FUNCTION_BLOCK "LGF_TimerSwitch"
{ S7_Optimized_Access := 'TRUE' }
VERSION : 0.1
   VAR_INPUT
      onMonth : USInt;   // Monat, in der der Ausgang gesetzt wird
      onDay : USInt;   // Tag, an dem der Ausgang gesetzt wird
      onWeekday : USInt;   // Wochentag, an dem der Ausgang gesetzt wird;  Sonntag: 1, Montag: 2, Dienstag: 3, ...
      onHour : USInt;   // Stunde, in der der Ausgang gesetzt wird
      onMinute : USInt;   // Minute, in der der Ausgang gesetzt wird
      offMonth : USInt;   // Monat, in der der Ausgang zurückgesetzt wird
      offDay : USInt;   // Tag, an dem der Ausgang zurückgesetzt wird
      offWeekday : USInt;   // Wochentag, an dem der Ausgang zurückgesetzt wird;  Sonntag: 1, Montag: 2, Dienstag: 3, ...
      offHour : USInt;   // Stunde, in der der Ausgang zurückgesetzt wird
      offMinute : USInt;   // Minute, in der der Ausgang zurückgesetzt wird
      mode : USInt;   // Angabe des Modus (siehe Funktionsweise);  Täglich: 1, Wöchentlich: 2, Monatlich: 3, Jährlich: 4, Arbeitstage: 5, Wochenende: 6
   END_VAR

   VAR_OUTPUT
      signal { ExternalWritable := 'False'} : Bool;   // Ausagngssignal
      actLocalTime {InstructionName := 'DTL'; LibVersion := '1.0'; ExternalWritable := 'False'} : DTL;   // Aktuelle Lokalzeit
      error { ExternalWritable := 'False'} : Bool;   // FALSE: Kein Fehler / TRUE: Während der Ausführung des FB ist ein Fehler aufgetreten
      status { ExternalWritable := 'False'} : Word;   // 16#0000-16#7FFF: Status des FB / 16#8000-16#FFFF: Fehleridentifikation (siehe folgende Tabelle)
      subFunctionStatus { ExternalWritable := 'False'} : Word;   // Status Word einer aufgerufenen Unterfunktion
   END_VAR

   VAR_TEMP
      tempTime {InstructionName := 'DTL'; LibVersion := '1.0'} : DTL;   // Temp Variable für die aktuelle Zeit und das aktuelle Datum von RD_LOC_T
      tempReadTimeStatus : Word;   // Status Wort der Systemfunktion RD_LOC_T
      tempOnTimeDtl {InstructionName := 'DTL'; LibVersion := '1.0'} : DTL;   // Temp Variable für Einschaltzeitpunkt (Zeit und Datum) DTL
      tempOnTimeTod : Time_Of_Day;   // Temp Variable für Einschaltzeitpunkt (Zeit) TOD
      tempOffTimeDtl {InstructionName := 'DTL'; LibVersion := '1.0'} : DTL;   // Temp Variable für Ausschaltzeitpunkt (Zeit und Datum) DTL
      tempOffTimeTod : Time_Of_Day;   // Temp Variable für Ausschaltzeitpunkt (Zeit) TOD
      tempActTimeDtl {InstructionName := 'DTL'; LibVersion := '1.0'} : DTL;   // Temp Variable für aktuelles Datum und aktuelle Zeit DTL
      tempActTimeTod : Time_Of_Day;   // Temp Variable für aktuelles Datum und aktuelle Zeit von RD_LOC_T / TOD
   END_VAR

   VAR CONSTANT
      ZERO : USInt := 0;   // Null Konstante zur Initialisierung
      CLEAR_DTL {InstructionName := 'DTL'; LibVersion := '1.0'} : DTL;   // Lösche Datum und Zeit mit leerer Varibale
      STATUS_NO_ERROR : Word := 16#0000;   // Status: kein Fehler aufgetreten
      ERR_NO_MODE_SELECTED : Word := 16#8200;   // Error: Kein vorhandener Mode ausgewählt, bitte Eingang `mode` prüfen
      ERR_RD_LOC_T : Word := 16#8600;   // Error in Funktion RD_LOC_T - weitere infos in `subFunctionStatus`
      MODE_DAILY : UInt := 1;   // Mode: Täglich
      MODE_WEEKLY : UInt := 2;   // Mode: Wöchentlich
      MODE_MONTHLY : UInt := 3;   // Mode: Monatlich
      MODE_YEARLY : UInt := 4;   // Mode: Jährlich
      MODE_WEEK_DAYS : UInt := 5;   // Mode: Wochentage
      MODE_WEEKEND_DAYS : UInt := 6;   // Mode: Wochenend Tage
      MONTH_JANUARY : USInt := 1;   // Monat Januar
      MONTH_DECEMBER : USInt := 12;   // Monat Dezember
      DAY_MONDAY : USInt := 2;   // Wochentag Montag
      DAY_FRIDAY : USInt := 6;   // Wochentag Freitag
      DAY_SATURDAY : USInt := 7;   // Wochentag Samstag
      DAY_SUNDAY : USInt := 1;   // Wochentag Sonntag
      DAY_NEXT_SUNDAY : USInt := 8;   // Wochentag - mächster Sonntag
      DAY_NEXT_MONDAY : USInt := 9;   // Wochentag - nächster Montag
      DATE_INCREMENT : USInt := 1;   // Inkremntierung für Datum (Monat oder Jahr)
      DAY_INCREMENT : Time := T#1d;   // Inkrementiere einen Tag
      WEEK_INCREMENT : Time := T#7d;   // Inkremntiere 7 Tage = 1 Woche
      DAYS_PER_WEEK : USInt := 7;   // Eine Woche = 7 Tage
      DEFAULT_YEAR : UInt := 2015;   // Default Jahr um im DTL Datentyp den Wochentag und das Datum zu synchronisieren
      DEFAULT_MONTH : USInt := 2;   // Default Monat um im DTL Datentyp den Wochentag und das Datum zu synchronisieren
   END_VAR


BEGIN
	REGION BLOCK INFO HEADER
	    //===============================================================================
	    // SIEMENS AG / (c)Copyright 2017
	    //-------------------------------------------------------------------------------
	    // Title:            LGF_TimerSwitch
	    // Comment/Function: Timer Switch (daily, weekly, monthly, working days, ...)
	    //                   Mode: Daily: 1, weekly: 2, monthly: 3, yearly: 4, workday: 5, weekend: 6
	    // Library/Family:   LGF(Library General Functions)
	    // Author:           Siemens Digital Industry Support
	    // Tested with:      CPU1212C DC/DC/DC FW:V4.2
	    // Engineering:      TIA Portal V14 Update 1
	    // Restrictions:     ENO disabled - error handling done with error and status
	    // Requirements:     PLC (S7-1200 / S7-1500)
	    //-------------------------------------------------------------------------------
	    // Change log table:
	    // Version  | Date       | Expert in charge       | Changes applied
	    //----------|------------|------------------------|------------------------------
	    // 01.00.00 19.08.2015  Siemens Industry Online Support
	    //                      First released version
	    // 01.00.01 16.11.2015  Siemens Industry Online Support
	    //                      Fix in mode 2
	    // 01.01.00 23.05.2016  Siemens Industry Online Support
	    //                      New mode 5 + 6
	    //                      New output: actLocalTime
	    // 01.01.01 02.01.2017  Siemens Industry Online Support
	    //                      Upgrade: TIA V14 Update 1
	    // 01.01.02 14.09.2018  Siemens Industry Online Support
	    //                      Fix in modes 1, 3, 5, 6
	    // 01.01.03 17.09.2018  Siemens Industry Online Support
	    //                      Upgrade: TIA V15 Update 2
	    // 01.01.04 10.10.2018  Siemens Industry Online Support
	    //                      Connection to type restored
	    // 01.01.05 23.11.2018  Siemens Industry Online Support
	    //                      Upgrade: TIA V15.1
	    // 01.01.10 13.11.2019  Simatic Systems Support
	    //                      Magic numbers removed, tag naming added, code reworked
	    // 03.00.00 23.04.2020  Simatic Systems Support
	    //                      Set version to V3.0.0, harmonize the version of the whole library
	    // 03.00.01 19.01.2020  Simatic Systems Support
	    //                      Insert documentation
	    //=============================================================================
	END_REGION BLOCK INFO HEADER

	REGION DESCRIPTION
	    (/*
	Hinweis
	:    In `subFunctionStatus` wird der Status von aufgerufenen Anweisungen ausge-geben. Der Ausgangswert in `status` gibt in diesem Fall an, welche Anweisung den Fehler verursacht hat. Holen Sie sich in diesem Fall die Informationen aus der TIA Portal Online Hilfe zu den jeweiligen Anweisungen.

	---

	Der Baustein bietet verschiedene Arten einer Zeitschaltuhr, die im Parameter `mode` bestimmt werden

	* Tägliche Zeitschaltuhr (mode = 1)
	* Wöchentliche Zeitschaltuhr (mode = 2)
	* Monatliche Zeitschaltuhr (mode = 3)
	* Jährliche Zeitschaltuhr (mode = 4)
	* Werktags, Montag bis Freitag (mode = 5)
	* Wochenende, Samstag und Sonntag (mode = 6)

	Der Zeitwert wird immer mit der Lokalzeit der SPS verglichen, daher muss der Zeitwert, der bei den On- und Off-Parametern angegeben wird, als lokale Zeit angegeben werden.

	Abhängig vom Modus müssen folgende Formalparameter beschaltet werden:

	+------+---------------------------------------+-----------------------------------------+
	| Mode | Mode                                  | Required formal parameters              |
	+======+=======================================+=========================================+
	| 1 .  | Tägliche Zeitschaltuhr                | * onHour / offHour                      |
	|      |                                       | * onMinute / offMinute                  |
	+------+---------------------------------------+-----------------------------------------+
	| 2 .  | Wöchentlich Zeitschaltuhr             | * onWeekday / offWeekday                |
	|      |                                       | * onHour / offHour                      |
	|      |                                       | * onMinute / offMinute                  |
	+------+---------------------------------------+-----------------------------------------+
	| 3 .  | Monatliche Zeitschaltuhr              | * onDay / offDay                        |
	|      |                                       | * onHour / offHour                      |
	|      |                                       | * onMinute / offMinute                  |
	+------+---------------------------------------+-----------------------------------------+
	| 4 .  | Jährliche Zeitschaltuhr               | * onMonth / offMonth                    |
	|      |                                       | * onDay / offDay                        |
	|      |                                       | * onHour / offHour                      |
	|      |                                       | * onMinute / offMinute                  |
	+------+---------------------------------------+-----------------------------------------+
	| 5 .  | Werktags                              | * onHour / offHour                      |
	|      |                                       | * onMinute / offMinute                  |
	+------+---------------------------------------+-----------------------------------------+
	| 6 .  | Wochenende                            | * onHour / offHour                      |
	|      |                                       | * onMinute / offMinute                  |
	+------+---------------------------------------+-----------------------------------------+

	Entspricht die eingestellte Startzeit der aktuellen Lokalzeit der Steuerung, wird der Ausgang `signal` auf `TRUE` gesetzt. Entspricht die eingestellte Abschaltzeit der aktuellen Lokalzeit der Steuerung, wird der Ausgang `signal` wieder zurückgesetzt.

	Hinweis
	:    Beachten Sie, dass der Baustein in den Modi „Monatliche Zeitschaltuhr“ (mode = 3) oder „Jährliche Zeitschaltuhr“ (mode = 4) nur dann schaltet, wenn die Tage, die Sie an den Eingangsparametern „onDay“ und „offDay“ angeben, tatsächlich in diesem Monat vorkommen.
	*/)
	END_REGION DESCRIPTION

	REGION INITIALISATION
	    // Time ON init
	    #tempOnTimeDtl.HOUR := #onHour;
	    #tempOnTimeDtl.MINUTE := #onMinute;
	    #tempOnTimeDtl.SECOND := #ZERO;
	    #tempOnTimeDtl.NANOSECOND := #ZERO;
	    // Time OFF init
	    #tempOffTimeDtl.HOUR := #offHour;
	    #tempOffTimeDtl.MINUTE := #offMinute;
	    #tempOffTimeDtl.SECOND := #ZERO;
	    #tempOffTimeDtl.NANOSECOND := #ZERO;
	END_REGION

	REGION READ LOCAL TIME
	    #tempReadTimeStatus := INT_TO_WORD(RD_LOC_T(#tempTime));

	    // check result for error --> 16#8000 / MSB .X15
	    IF #tempReadTimeStatus.%X15 THEN
	        #error := TRUE;
	        #status := #ERR_RD_LOC_T;
	        #subFunctionStatus := #tempReadTimeStatus;
	        #actLocalTime := #CLEAR_DTL;
	        #signal := FALSE;
	        RETURN;
	    END_IF;

	    // Store time of the current day
	    #tempActTimeDtl := #tempTime;
	    #tempActTimeTod := DTL_TO_TOD(#tempTime);
	END_REGION

	REGION TIMER SWITCH LOGIC
	    CASE #mode OF
	        #MODE_DAILY:
	            REGION DAILY MODE
	                #tempOnTimeDtl.YEAR := #tempActTimeDtl.YEAR;
	                #tempOnTimeDtl.MONTH := #tempActTimeDtl.MONTH;
	                #tempOnTimeDtl.WEEKDAY := #tempActTimeDtl.WEEKDAY;
	                #tempOnTimeDtl.DAY := #tempActTimeDtl.DAY;
	                // Store time of the on day
	                #tempOnTimeTod := DTL_TO_TOD(#tempOnTimeDtl);

	                #tempOffTimeDtl.YEAR := #tempActTimeDtl.YEAR;
	                #tempOffTimeDtl.MONTH := #tempActTimeDtl.MONTH;
	                #tempOffTimeDtl.WEEKDAY := #tempActTimeDtl.WEEKDAY;
	                #tempOffTimeDtl.DAY := #tempActTimeDtl.DAY;
	                // Store time of the off day
	                #tempOffTimeTod := DTL_TO_TOD(#tempOffTimeDtl);

	                // Timer setting - overnight
	                IF #tempOnTimeTod > #tempOffTimeTod THEN
	                    // Increase the day of the timeOff when midnight happens
	                    IF #tempActTimeTod > #tempOffTimeTod THEN
	                        #tempOffTimeDtl := #tempOffTimeDtl + #DAY_INCREMENT;
	                    ELSE
	                        // Decrease the day of the timeOn when midnight happens
	                        // Activate signal from the midnight
	                        #tempOnTimeDtl := #tempOnTimeDtl - #DAY_INCREMENT;
	                    END_IF;
	                END_IF;
	            END_REGION

	        #MODE_WEEKLY:
	            REGION WEEKLY MODE
	                // Set the default date
	                #tempOnTimeDtl.YEAR := #DEFAULT_YEAR;
	                #tempOnTimeDtl.MONTH := #DEFAULT_MONTH;
	                #tempOnTimeDtl.DAY := #onWeekday;  // Synchronize DTL.WEEKDAY with date

	                #tempOnTimeTod := DTL_TO_TOD(#tempOnTimeDtl);

	                #tempOffTimeDtl.YEAR := #DEFAULT_YEAR;
	                #tempOffTimeDtl.MONTH := #DEFAULT_MONTH;
	                #tempOffTimeDtl.DAY := #offWeekday;

	                #tempOffTimeTod := DTL_TO_TOD(#tempOffTimeDtl);

	                #tempActTimeDtl.YEAR := #DEFAULT_YEAR;
	                #tempActTimeDtl.MONTH := #DEFAULT_MONTH;
	                #tempActTimeDtl.DAY := #tempActTimeDtl.WEEKDAY;

	                IF #onWeekday > #offWeekday OR
	                    (#onWeekday = #offWeekday AND #tempOnTimeTod > #tempOffTimeTod) THEN
	                    #tempOffTimeDtl.DAY := #offWeekday + #DAYS_PER_WEEK;

	                    IF #onWeekday > #tempActTimeDtl.WEEKDAY OR
	                        (#onWeekday = #offWeekday AND #tempActTimeTod < #tempOffTimeTod) THEN
	                        #tempActTimeDtl.DAY := #tempActTimeDtl.WEEKDAY + #DAYS_PER_WEEK;
	                    END_IF;
	                END_IF;
	            END_REGION

	        #MODE_MONTHLY:
	            REGION MONTHLY MODE
	                #tempOnTimeDtl.YEAR := #tempActTimeDtl.YEAR;
	                #tempOnTimeDtl.MONTH := #tempActTimeDtl.MONTH;
	                #tempOnTimeDtl.WEEKDAY := #tempActTimeDtl.WEEKDAY;
	                #tempOnTimeDtl.DAY := #onDay;

	                #tempOnTimeTod := DTL_TO_TOD(#tempOnTimeDtl);

	                #tempOffTimeDtl.YEAR := #tempActTimeDtl.YEAR;
	                #tempOffTimeDtl.MONTH := #tempActTimeDtl.MONTH;
	                #tempOffTimeDtl.WEEKDAY := #tempActTimeDtl.WEEKDAY;
	                #tempOffTimeDtl.DAY := #offDay;

	                #tempOffTimeTod := DTL_TO_TOD(#tempOffTimeDtl);

	                // Timer setting - over new year
	                IF #onDay > #offDay OR
	                    (#onDay = #offDay AND #tempOnTimeTod > #tempOffTimeTod) THEN
	                    IF #tempActTimeDtl.DAY > #offDay OR
	                        (#tempActTimeDtl.DAY = #offDay AND #tempActTimeTod > #tempOffTimeTod) THEN
	                        // Increase the month of the timeOff over new year
	                        IF #tempOffTimeDtl.MONTH = #MONTH_DECEMBER THEN
	                            #tempOffTimeDtl.MONTH := #MONTH_JANUARY;
	                            #tempOffTimeDtl.YEAR := #tempOffTimeDtl.YEAR + #DATE_INCREMENT;
	                        ELSE
	                            #tempOffTimeDtl.MONTH := #tempOffTimeDtl.MONTH + #DATE_INCREMENT;
	                        END_IF;
	                    ELSE
	                        // Decrease the month of the timeOn over new year
	                        IF #tempOnTimeDtl.MONTH = #MONTH_JANUARY THEN
	                            #tempOnTimeDtl.MONTH := #MONTH_DECEMBER;
	                            #tempOnTimeDtl.YEAR := #tempOnTimeDtl.YEAR - #DATE_INCREMENT;
	                        ELSE
	                            #tempOnTimeDtl.MONTH := #tempOnTimeDtl.MONTH - #DATE_INCREMENT;
	                        END_IF;

	                    END_IF;
	                END_IF;
	            END_REGION

	        #MODE_YEARLY:
	            REGION YEARLY MODE
	                #tempOnTimeDtl.YEAR := #tempActTimeDtl.YEAR;
	                #tempOnTimeDtl.MONTH := #onMonth;
	                #tempOnTimeDtl.WEEKDAY := #tempActTimeDtl.WEEKDAY;
	                #tempOnTimeDtl.DAY := #onDay;

	                #tempOnTimeTod := DTL_TO_TOD(#tempOnTimeDtl);

	                #tempOffTimeDtl.YEAR := #tempActTimeDtl.YEAR;
	                #tempOffTimeDtl.MONTH := #offMonth;
	                #tempOffTimeDtl.WEEKDAY := #tempActTimeDtl.WEEKDAY;
	                #tempOffTimeDtl.DAY := #offDay;

	                #tempOffTimeTod := DTL_TO_TOD(#tempOffTimeDtl);

	                // Timer setting - over new year
	                IF #onMonth > #offMonth OR
	                    (#onMonth = #offMonth AND #tempOnTimeTod > #tempOffTimeTod) THEN
	                    IF #tempActTimeDtl.MONTH > #offMonth OR
	                        (#tempActTimeDtl.MONTH = #offMonth AND #tempActTimeTod > #tempOffTimeTod) THEN
	                        // Increase the year of the timeOff when new year happens
	                        #tempOffTimeDtl.YEAR := #tempOffTimeDtl.YEAR + #DATE_INCREMENT;
	                    ELSE
	                        // Decrease the year of the timeOn when new year happens
	                        #tempOnTimeDtl.YEAR := #tempOnTimeDtl.YEAR - #DATE_INCREMENT;
	                    END_IF;
	                END_IF;
	            END_REGION

	        #MODE_WEEK_DAYS:  // Working days (Monday - Friday)
	            REGION WEEK DAYS MODE
	                #tempOnTimeDtl.YEAR := #DEFAULT_YEAR;
	                #tempOnTimeDtl.MONTH := #DEFAULT_MONTH;
	                #tempOnTimeDtl.DAY := #tempActTimeDtl.WEEKDAY;

	                #tempOnTimeTod := DTL_TO_TOD(#tempOnTimeDtl);

	                #tempOffTimeDtl.YEAR := #DEFAULT_YEAR;
	                #tempOffTimeDtl.MONTH := #DEFAULT_MONTH;
	                #tempOffTimeDtl.DAY := #tempActTimeDtl.WEEKDAY;

	                #tempOffTimeTod := DTL_TO_TOD(#tempOffTimeDtl);

	                #tempActTimeDtl.YEAR := #DEFAULT_YEAR;
	                #tempActTimeDtl.MONTH := #DEFAULT_MONTH;
	                #tempActTimeDtl.DAY := #tempActTimeDtl.WEEKDAY;

	                // Timer setting - overnight
	                IF #tempOnTimeTod > #tempOffTimeTod THEN
	                    IF #tempActTimeTod > #tempOffTimeTod THEN
	                        #tempOffTimeDtl := #tempOffTimeDtl + #DAY_INCREMENT;
	                    ELSE
	                        #tempOnTimeDtl := #tempOnTimeDtl - #DAY_INCREMENT;
	                    END_IF;
	                END_IF;

	                IF #tempOnTimeDtl.DAY <= #DAY_MONDAY THEN
	                    #tempOnTimeDtl.DAY := #DAY_MONDAY;
	                ELSIF #tempOnTimeDtl.DAY > #DAY_FRIDAY THEN
	                    #tempOnTimeDtl.DAY := #DAY_FRIDAY;
	                END_IF;

	                IF #tempOffTimeDtl.DAY > #DAY_FRIDAY AND
	                    #tempOnTimeTod > #tempOffTimeTod THEN // #tempOffTime > Friday AND crossed midnight
	                    #tempOffTimeDtl.DAY := #DAY_SATURDAY;
	                ELSIF #tempOffTimeDtl.DAY > #DAY_FRIDAY THEN
	                    #tempOffTimeDtl.DAY := #DAY_FRIDAY;
	                END_IF;
	            END_REGION

	        #MODE_WEEKEND_DAYS:  // Weekend (Saturday and Sunday)
	            REGION WEEKEND DAYS MODE
	                #tempOnTimeDtl.YEAR := #DEFAULT_YEAR;
	                #tempOnTimeDtl.MONTH := #DEFAULT_MONTH;
	                #tempOnTimeDtl.DAY := #tempActTimeDtl.WEEKDAY;

	                IF #tempOnTimeDtl.DAY < #DAY_SATURDAY THEN
	                    #tempOnTimeDtl := #tempOnTimeDtl + #WEEK_INCREMENT;
	                END_IF;

	                #tempOnTimeTod := DTL_TO_TOD(#tempOnTimeDtl);

	                #tempOffTimeDtl.YEAR := #DEFAULT_YEAR;
	                #tempOffTimeDtl.MONTH := #DEFAULT_MONTH;
	                #tempOffTimeDtl.DAY := #tempActTimeDtl.WEEKDAY;

	                IF #tempOffTimeDtl.DAY < #DAY_SATURDAY THEN
	                    #tempOffTimeDtl := #tempOffTimeDtl + #WEEK_INCREMENT;
	                END_IF;

	                #tempOffTimeTod := DTL_TO_TOD(#tempOffTimeDtl);

	                #tempActTimeDtl.YEAR := #DEFAULT_YEAR;
	                #tempActTimeDtl.MONTH := #DEFAULT_MONTH;
	                #tempActTimeDtl.DAY := #tempActTimeDtl.WEEKDAY;

	                IF #tempActTimeDtl.DAY < #DAY_SATURDAY THEN
	                    #tempActTimeDtl := #tempActTimeDtl + #WEEK_INCREMENT;
	                END_IF;

	                #tempActTimeTod := DTL_TO_TOD(#tempTime);

	                // Timer setting - overnight
	                IF #tempOnTimeTod > #tempOffTimeTod THEN
	                    IF #tempActTimeTod > #tempOffTimeTod THEN
	                        #tempOffTimeDtl := #tempOffTimeDtl + #DAY_INCREMENT;
	                    ELSE
	                        #tempOnTimeDtl := #tempOnTimeDtl - #DAY_INCREMENT;
	                    END_IF;
	                END_IF;

	                IF #tempOnTimeDtl.DAY < #DAY_SATURDAY THEN
	                    #tempOnTimeDtl.DAY := #DAY_SATURDAY;
	                ELSIF #tempOnTimeDtl.DAY > #DAY_NEXT_SUNDAY THEN
	                    #tempOnTimeDtl.DAY := #DAY_NEXT_SUNDAY;
	                END_IF;

	                IF #tempOffTimeDtl.DAY > #DAY_NEXT_SUNDAY AND
	                    #tempOnTimeTod > #tempOffTimeTod THEN // #tempOffTime.DAY > Sunday AND crossed midnight
	                    #tempOffTimeDtl.DAY := #DAY_NEXT_MONDAY;
	                ELSIF #tempOffTimeDtl.DAY > #DAY_NEXT_SUNDAY THEN
	                    #tempOffTimeDtl.DAY := #DAY_NEXT_SUNDAY;
	                END_IF;
	            END_REGION
	        ELSE
	            #signal := FALSE;
	            #actLocalTime := #CLEAR_DTL;
	            #error := TRUE;
	            #status := #ERR_NO_MODE_SELECTED;
	            #subFunctionStatus := USINT_TO_WORD(#mode);
	            RETURN;
	    END_CASE;

	END_REGION

	REGION OUTPUT
	    #actLocalTime := #tempTime;
	    #signal := (#tempActTimeDtl >= #tempOnTimeDtl) AND (#tempActTimeDtl < #tempOffTimeDtl);
	    #error := false;
	    #status := #STATUS_NO_ERROR;
	    #subFunctionStatus := #STATUS_NO_ERROR;

	    // ENO is not used, forced to TRUE
	    ENO := TRUE;
	END_REGION

END_FUNCTION_BLOCK

